TYPE ST_BigBagActualMassStoreStatus :
STRUCT
    sDiag : T_MaxString;
END_STRUCT
END_TYPE

(* stored: Version 1.1.0.1, ProductVersion 3.1.4024.16
   DUT ST_BigBagActualMassStoreStatus: Id {6f08aadc-6cff-4dbe-972f-ba58169a2ace} *)
